FUNCTION_BLOCK EL4104
VAR
	_io : EL4xx4_Data;
	{attribute addProperty Name "WcState"}
	_wcState : WcStateBase;
	{attribute addProperty Name "Info data"}
	_infoData : InfoDataAds;
END_VAR

PROPERTY IO : REFERENCE TO EL4xx4_Data
GET
IO REF= _io;
END_GET
END_PROPERTY

PROPERTY WcState : REFERENCE TO WcStateBase
GET
WcState REF= _wcState;
END_GET
END_PROPERTY

END_FUNCTION_BLOCK

(* stored: Version 1.1.0.1, ProductVersion 3.1.4024.9
   POU EL4104: Id {0ad071d4-c870-036e-22ce-28830724c2b2}, SpecialFunc None
   Property IO: Id {e77b2814-4404-0f2a-2a5b-a05677860919}
   Get Get: Id {6ed950d5-ecf6-0cff-0248-479e921acc16}
   Property WcState: Id {dd0a6108-12cb-0ce2-3a17-4054ccc42ecb}
   Get Get: Id {defd9c6e-69a4-07d8-39b7-d6e9f200726d} *)
